Staubli VAL3: loadPage.pgx

program loadPage(string x_sPage, string& x_sItems[])
// load the next page
  local num i
  local string l_sMessage
  local num l_nClock
begin
  // look if the page libload is correct
  i=page:libLoad(x_sPage)
  if i!=0
    logMsg("[VALlaser] INTERFACE:PAGE LIBLOAD "+x_sPage+" result "+toString("",i))
    call language:message(l_sMessage,-7)
    popUpMsg(l_sMessage+x_sPage+" ; "+toString("",i))
  else
    // copy all the field from x_sItems to the next page
    call use:stringCopy(x_sItems,page:sItems)
    call page:main()
    // to give back
    call use:stringCopy(page:sItems,x_sItems)
  endIf
end
